TYPE "IPC_Msg_Generico"
VERSION : 0.1
// Block: IPC_Msg_Generico
   STRUCT
      Id : DInt;
      timestamp : String;
      topic : UDInt;
      payLoad : String;
   END_STRUCT;

END_TYPE
